# EPICS autosave request: iocBoot/sioc-esb-thfw01/thorFW.req
$(P):POS:SC.ZRST
$(P):POS:SC.ONST
$(P):POS:SC.TWST
$(P):POS:SC.THST
$(P):POS:SC.FRST
$(P):POS:SC.FVST
